PROGRAM myParts
VAR
END_VAR

END_PROGRAM

(* stored: Version 1.1.0.1, ProductVersion 3.1.4024.11
   POU myParts: Id {644fb9b2-df71-440f-9e4f-905e2e095be0}, SpecialFunc None *)
